Fanuc KAREL source: kc00005.KL

-- PROVISIONAL review KL for V940-1; original PC SHA256 858f0e4f15663fc2840a23327551a37c2eb9a6aefda2f5780db5633a3016eb8a
-- Incomplete behavior may be omitted. Consult companion uncertainty JSON. Do not deploy.
PROGRAM KC00005
%NOLOCKGROUP
BEGIN
  -- V9_ZERO_TABLE_METADATA_HINT layout=0002_ascii; no indexed target words; source/name/runtime held
  -- UNRESOLVED_PC offsets 5-27; opcodes 27,22,22,22,31
  -- UNRESOLVED_PC offsets 32-36; opcodes 7F
END KC00005
